FUNCTION_BLOCK FB_DiagnosisEtherCATMaster
VAR_OUTPUT
	bError						:BOOL;								//エラー発生を出力
END_VAR
VAR_IN_OUT
	fbFrmWcStateDiagnosis		:ARRAY[*] OF FB_FrmWcStateDiagnosis;
	fbFrmStateDiagnosis			:ARRAY[*] OF FB_FrmStateDiagnosis;
END_VAR
VAR
	_eEtherCATMaster			:E_EtherCATMaster;	

	fbDevStateDiagnosis			:FB_DevStateDiagnosis;
	fbSlaveCountDiagnosis		:FB_SlaveCountDiagnosis;
	i							:DINT;
END_VAR

//診断用FBを呼び出し
fbDevStateDiagnosis(eEtherCATMaster:=_eEtherCATMaster);
fbSlaveCountDiagnosis(eEtherCATMaster:=_eEtherCATMaster);

bError:=fbDevStateDiagnosis.bError OR fbSlaveCountDiagnosis.bError;

//可変長のアレイを診断と出力
FOR i := LOWER_BOUND(fbFrmWcStateDiagnosis,1) TO UPPER_BOUND(fbFrmWcStateDiagnosis,1) DO
	fbFrmWcStateDiagnosis[i](eEtherCATMaster:=_eEtherCATMaster);
	bError:=bError OR fbFrmWcStateDiagnosis[i].bError;
END_FOR

FOR i := LOWER_BOUND(fbFrmStateDiagnosis,1) TO UPPER_BOUND(fbFrmStateDiagnosis,1) DO
	fbFrmStateDiagnosis[i](eEtherCATMaster:=_eEtherCATMaster);
	bError:=bError OR fbFrmStateDiagnosis[i].bError;
END_FOR

//FB_Init は常に暗黙的に使用可能で、主に初期化に使用されます。
//戻り値は評価されません。特定の結果を得るために、メソッドを明示的に宣言し、
//そのメソッドに標準の初期化コードをもったコードを追加することができます。戻り値を評価できます。
METHOD FB_Init: BOOL
VAR_INPUT
    bInitRetains: BOOL; // TRUE: 保持変数は初期化されます (ウォーム リセット、あるいはコールド リセット)
    bInCopyCode: BOOL;  // TRUE: 後でコードをコピーする (オンライン変更) ために、インスタンスをコピーします。
	
	eEtherCATMaster	:E_EtherCATMaster;
END_VAR
_eEtherCATMaster:=eEtherCATMaster;
END_METHOD

END_FUNCTION_BLOCK

(* stored: Version 1.1.0.1, ProductVersion 3.1.4026.18
   POU FB_DiagnosisEtherCATMaster: Id {de43cf2f-fd79-46c9-9b8b-af34aac85cac}, SpecialFunc None
   Method FB_Init: Id {f96e1ce9-536b-48ad-ae01-8a8fafddca42} *)
